// TIA Portal V20 export
TYPE "Station"
   STRUCT
      SensorA : Bool;
      SensorB : Bool;
      SensorC : Bool;
      SensorD : Bool;
      isEmpty : Bool;
      isOccupied : Bool;
   END_STRUCT;
END_TYPE
